RoboDK station: AmbienteRecriado.rdk

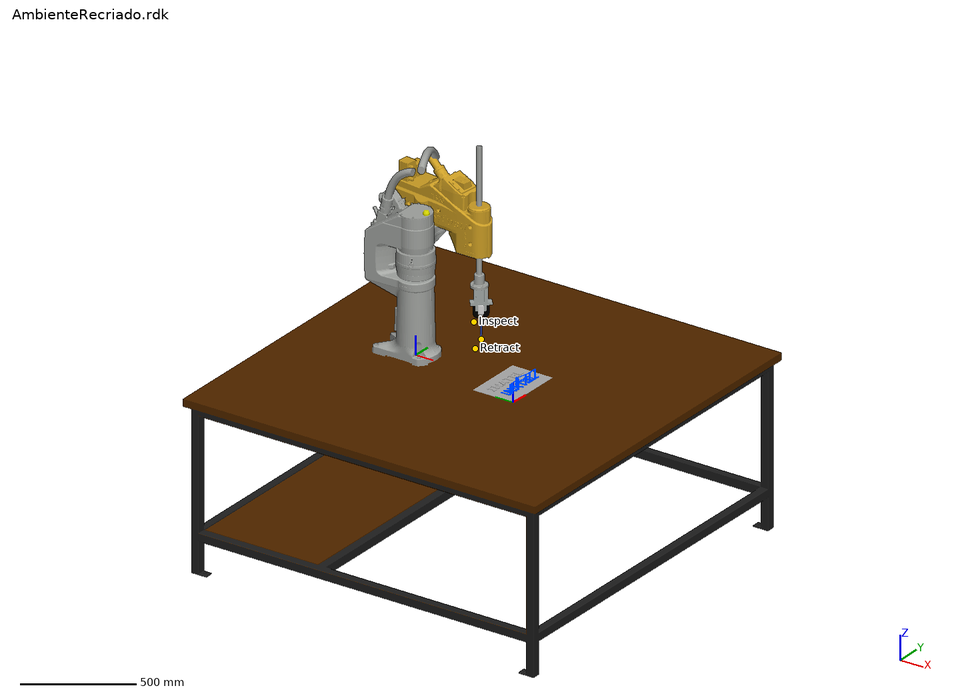
[picture v0: the station drawn from its stored meshes, robots at their saved joint values, targets as dots, program paths as lines]
Station FollowCurves_Inatel (saved by RoboDK 5.5.2). Poses are relative to the parent item; angles as X-Y-Z fixed-axis rotations.
  - frame World at (0, 0, 835) mm
    - robot Staubli TS60 FL 200 (model Staubli TS60 FL 400): 4 axes, payload 2 kg, reach 600 mm, repeatability 0.01 mm, weight 55 kg
        modified DH rows (alpha deg, a mm, theta deg, d mm): 0, 0, 0, 0; 0, 330, 0, 0; 0, 270, 0, 170 linear; 180, 0, 0, 0
        joint limits [-140, -150, 0, -500] to [140, 150, 200, 500]; home [0, 0, 0, 0]; saved at [112.244, -119.359, 90, 172.885]
      - tool GarraCompleta, TCP at (0, 0, 200) mm, size 97 x 40 x 153.1 mm, geometry from GarraCompleta.STL
        - object Suporte_e_Caneta at (4.39, 18.92, -137) mm, rotated rx 0 ry 0 rz 48 deg, size 26 x 26 x 165.9 mm, geometry from Suporte_e_Caneta.STL
      - tool TCP_Garra, TCP at (0, 17, 260) mm
    - frame Reference SW at (610, -140, 0) mm, rotated rx 0 ry 0 rz 90 deg
      - object SWPart at (0, 0, 0) mm, size 295 x 210 x 6 mm, geometry from SWPart.stl
    - target Retract (Cartesian target) at (261.87, 75.71, 73.19) mm, rotated rx -180 ry 0 rz 180 deg; joints [65.057, -128.028, 163.19, 117.03] of Staubli TS60 FL 200
    - target Inspect (Cartesian target) at (104.05, 290.73, 73.19) mm, rotated rx -180 ry 0 rz -180 deg; joints [120.14, -122.614, 163.19, 177.527] of Staubli TS60 FL 200
    - target Peça (Cartesian target) at (143, 289, 0) mm, rotated rx -180 ry 0 rz -180 deg; joints [120.14, -122.614, 163.19, 177.527] of Staubli TS60 FL 200
    - target Encaixe (Cartesian target) at (143, 289, 0) mm, rotated rx -180 ry 0 rz -180 deg; joints [120.14, -122.614, 163.19, 177.527] of Staubli TS60 FL 200
  - object Mesa at (350, 0, 0) mm, size 1850 x 1850 x 835 mm, geometry from Mesa.STL
  - program Attach (1 instructions, listed below)
  - machining project Path1 settings: rotZ(0) | rotX(0)*rotY(0) | rotz(0) | onStart | onPathStart | onApproach | onPoint | onRetract | onFinish | SetRPM(%1) | SetTool(%1) | Extruder(%1) | default | default | OutOnMov(%1) | OutOffMov(%1) | onPathFinish | M_RunCode(%1)
  - program Path1 (314 instructions, listed below)
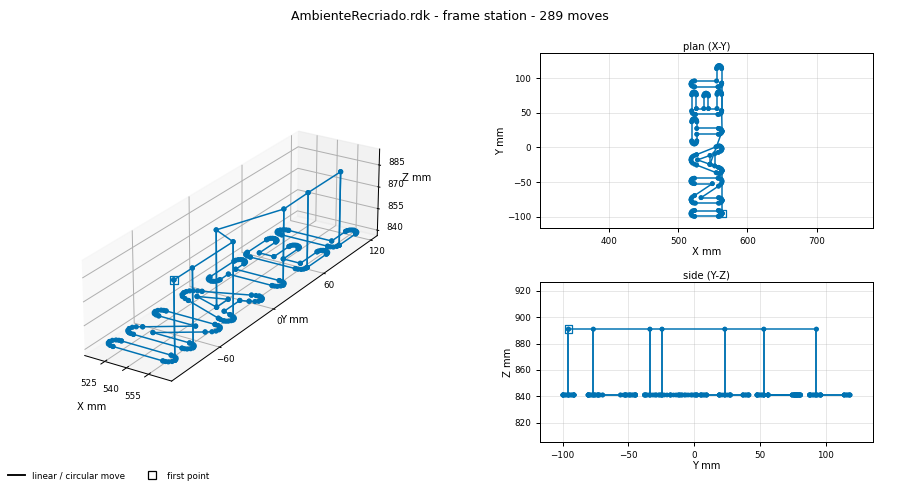
[picture p0: tool path of AmbienteRecriado.rdk in frame station, 289 of 289 moves have a stored position in this frame; points joined in program order, loops and branches not executed]

--- program Attach (robot Staubli TS60 FL 200) ---
  Attach to GarraCompleta

--- program Path1 (robot Staubli TS60 FL 200) ---
  Smooth(1)
  Set speed (1000.0 mm/s)
  Set Ref.: Reference SW
  Set Tool: TCP_Garra
  Show TCP_Garra
  MoveJ 1 to (44.52, 46.68, 56) mm, rotated rx -180 ry 0 rz 90 deg; joints [3.841, -33.741, 146, 150.101]
  MoveL 2 to (44.52, 46.68, 56) mm, rotated rx -180 ry 0 rz 90 deg; joints [3.841, -33.741, 146, 150.101]
  MoveL 3 to (44.52, 46.68, 6) mm, rotated rx -180 ry 0 rz 90 deg; joints [3.841, -33.741, 96, 150.101]
  MoveL 4 to (44.52, 46.68, 6) mm, rotated rx -180 ry 0 rz 90 deg; joints [3.841, -33.741, 96, 150.101]
  Set speed (50.0 mm/s)
  MoveL 5 to (42.47, 47.22, 6) mm, rotated rx -180 ry 0 rz 90 deg; joints [3.667, -33.825, 96, 149.843]
  MoveL 6 to (41.01, 48.77, 6) mm, rotated rx -180 ry 0 rz 90 deg; joints [3.851, -34.627, 96, 149.224]
  MoveL 7 to (40.48, 50.37, 6) mm, rotated rx -180 ry 0 rz 90 deg; joints [4.183, -35.562, 96, 148.621]
  MoveL 8 to (40.34, 52.05, 6) mm, rotated rx -180 ry 0 rz 90 deg; joints [4.583, -36.569, 96, 148.014]
  MoveL 9 to (40.34, 52.05, 6) mm, rotated rx -180 ry 0 rz 90 deg; joints [4.583, -36.569, 96, 148.014]
  MoveL 10 to (40.34, 86.33, 6) mm, rotated rx -180 ry 0 rz 90 deg; joints [11.299, -53.485, 96, 137.814]
  MoveL 11 to (40.34, 86.33, 6) mm, rotated rx -180 ry 0 rz 90 deg; joints [11.299, -53.485, 96, 137.814]
  MoveL 12 to (40.58, 88.46, 6) mm, rotated rx -180 ry 0 rz 90 deg; joints [11.67, -54.391, 96, 137.279]
  MoveL 13 to (41.53, 90.37, 6) mm, rotated rx -180 ry 0 rz 90 deg; joints [12.104, -55.258, 96, 136.846]
  MoveL 14 to (42.87, 91.36, 6) mm, rotated rx -180 ry 0 rz 90 deg; joints [12.451, -55.78, 96, 136.67]
  MoveL 15 to (44.52, 91.68, 6) mm, rotated rx -180 ry 0 rz 90 deg; joints [12.736, -56.054, 96, 136.682]
  MoveL 16 to (44.52, 91.68, 6) mm, rotated rx -180 ry 0 rz 90 deg; joints [12.736, -56.054, 96, 136.682]
  MoveL 17 to (46.6, 91.17, 6) mm, rotated rx -180 ry 0 rz 90 deg; joints [12.956, -56.028, 96, 136.929]
  MoveL 18 to (48.1, 89.64, 6) mm, rotated rx -180 ry 0 rz 90 deg; joints [12.935, -55.538, 96, 137.397]
  MoveL 19 to (48.65, 88.03, 6) mm, rotated rx -180 ry 0 rz 90 deg; joints [12.762, -54.929, 96, 137.833]
  MoveL 20 to (48.78, 86.33, 6) mm, rotated rx -180 ry 0 rz 90 deg; joints [12.512, -54.24, 96, 138.272]
  MoveL 21 to (48.78, 86.33, 6) mm, rotated rx -180 ry 0 rz 90 deg; joints [12.512, -54.24, 96, 138.272]
  MoveL 22 to (48.78, 52.05, 6) mm, rotated rx -180 ry 0 rz 90 deg; joints [5.865, -37.581, 96, 148.284]
  MoveL 23 to (48.78, 52.05, 6) mm, rotated rx -180 ry 0 rz 90 deg; joints [5.865, -37.581, 96, 148.284]
  MoveL 24 to (48.55, 49.89, 6) mm, rotated rx -180 ry 0 rz 90 deg; joints [5.298, -36.265, 96, 149.033]
  MoveL 25 to (47.57, 47.97, 6) mm, rotated rx -180 ry 0 rz 90 deg; joints [4.657, -34.958, 96, 149.699]
  MoveL 26 to (46.19, 46.99, 6) mm, rotated rx -180 ry 0 rz 90 deg; joints [4.184, -34.157, 96, 150.027]
  MoveL 27 to (44.52, 46.68, 6) mm, rotated rx -180 ry 0 rz 90 deg; joints [3.841, -33.741, 96, 150.101]
  Set speed (1000.0 mm/s)
  MoveL 28 to (44.52, 46.68, 6) mm, rotated rx -180 ry 0 rz 90 deg; joints [3.841, -33.741, 96, 150.101]
  MoveL 29 to (44.52, 46.68, 56) mm, rotated rx -180 ry 0 rz 90 deg; joints [3.841, -33.741, 146, 150.101]
  Set speed (1000.0 mm/s)
  MoveL 30 to (63.41, 46.68, 56) mm, rotated rx -180 ry 0 rz 90 deg; joints [6.675, -35.932, 146, 150.744]
  MoveL 31 to (63.41, 46.68, 6) mm, rotated rx -180 ry 0 rz 90 deg; joints [6.675, -35.932, 96, 150.744]
  MoveL 32 to (63.41, 46.68, 6) mm, rotated rx -180 ry 0 rz 90 deg; joints [6.675, -35.932, 96, 150.744]
  Set speed (50.0 mm/s)
  MoveL 33 to (61.47, 47.18, 6) mm, rotated rx -180 ry 0 rz 90 deg; joints [6.523, -36.039, 96, 150.484]
  MoveL 34 to (60.1, 48.64, 6) mm, rotated rx -180 ry 0 rz 90 deg; joints [6.695, -36.785, 96, 149.91]
  MoveL 35 to (59.6, 50.14, 6) mm, rotated rx -180 ry 0 rz 90 deg; joints [6.995, -37.63, 96, 149.365]
  MoveL 36 to (59.47, 51.72, 6) mm, rotated rx -180 ry 0 rz 90 deg; joints [7.358, -38.539, 96, 148.819]
  MoveL 37 to (59.47, 51.72, 6) mm, rotated rx -180 ry 0 rz 90 deg; joints [7.358, -38.539, 96, 148.819]
  MoveL 38 to (59.47, 85.3, 6) mm, rotated rx -180 ry 0 rz 90 deg; joints [13.85, -54.68, 96, 139.171]
  MoveL 39 to (59.47, 85.3, 6) mm, rotated rx -180 ry 0 rz 90 deg; joints [13.85, -54.68, 96, 139.171]
  MoveL 40 to (59.58, 87.2, 6) mm, rotated rx -180 ry 0 rz 90 deg; joints [14.17, -55.47, 96, 138.7]
  MoveL 41 to (59.93, 88.65, 6) mm, rotated rx -180 ry 0 rz 90 deg; joints [14.447, -56.087, 96, 138.36]
  MoveL 42 to (59.93, 88.65, 6) mm, rotated rx -180 ry 0 rz 90 deg; joints [14.447, -56.087, 96, 138.36]
  MoveL 43 to (60.79, 90.01, 6) mm, rotated rx -180 ry 0 rz 90 deg; joints [14.778, -56.697, 96, 138.08]
  MoveL 44 to (62.05, 91.02, 6) mm, rotated rx -180 ry 0 rz 90 deg; joints [15.107, -57.19, 96, 137.917]
  MoveL 45 to (64.47, 91.68, 6) mm, rotated rx -180 ry 0 rz 90 deg; joints [15.542, -57.625, 96, 137.918]
  MoveL 46 to (64.47, 91.68, 6) mm, rotated rx -180 ry 0 rz 90 deg; joints [15.542, -57.625, 96, 137.918]
  MoveL 47 to (66.75, 91.13, 6) mm, rotated rx -180 ry 0 rz 90 deg; joints [15.773, -57.568, 96, 138.204]
  MoveL 48 to (68.49, 89.54, 6) mm, rotated rx -180 ry 0 rz 90 deg; joints [15.764, -57.054, 96, 138.71]
  MoveL 49 to (70.49, 86.4, 6) mm, rotated rx -180 ry 0 rz 90 deg; joints [15.541, -55.923, 96, 139.618]
  MoveL 50 to (70.49, 86.4, 6) mm, rotated rx -180 ry 0 rz 90 deg; joints [15.541, -55.923, 96, 139.618]
  MoveL 51 to (87.59, 60.74, 6) mm, rotated rx -180 ry 0 rz 90 deg; joints [13.186, -45.589, 96, 147.597]
  MoveL 52 to (87.59, 60.74, 6) mm, rotated rx -180 ry 0 rz 90 deg; joints [13.186, -45.589, 96, 147.597]
  MoveL 53 to (87.59, 86.63, 6) mm, rotated rx -180 ry 0 rz 90 deg; joints [17.859, -57.048, 96, 140.811]
  MoveL 54 to (87.59, 86.63, 6) mm, rotated rx -180 ry 0 rz 90 deg; joints [17.859, -57.048, 96, 140.811]
  MoveL 55 to (87.81, 88.64, 6) mm, rotated rx -180 ry 0 rz 90 deg; joints [18.205, -57.858, 96, 140.348]
  MoveL 56 to (88.67, 90.44, 6) mm, rotated rx -180 ry 0 rz 90 deg; joints [18.602, -58.614, 96, 139.989]
  MoveL 57 to (89.94, 91.38, 6) mm, rotated rx -180 ry 0 rz 90 deg; joints [18.913, -59.045, 96, 139.869]
  MoveL 58 to (91.49, 91.68, 6) mm, rotated rx -180 ry 0 rz 90 deg; joints [19.161, -59.236, 96, 139.925]
  MoveL 59 to (91.49, 91.68, 6) mm, rotated rx -180 ry 0 rz 90 deg; joints [19.161, -59.236, 96, 139.925]
  MoveL 60 to (93.45, 91.21, 6) mm, rotated rx -180 ry 0 rz 90 deg; joints [19.342, -59.147, 96, 140.195]
  MoveL 61 to (94.84, 89.75, 6) mm, rotated rx -180 ry 0 rz 90 deg; joints [19.294, -58.644, 96, 140.65]
  MoveL 62 to (95.34, 88.23, 6) mm, rotated rx -180 ry 0 rz 90 deg; joints [19.118, -58.07, 96, 141.048]
  MoveL 63 to (95.47, 86.63, 6) mm, rotated rx -180 ry 0 rz 90 deg; joints [18.879, -57.442, 96, 141.437]
  MoveL 64 to (95.47, 86.63, 6) mm, rotated rx -180 ry 0 rz 90 deg; joints [18.879, -57.442, 96, 141.437]
  MoveL 65 to (95.47, 52.41, 6) mm, rotated rx -180 ry 0 rz 90 deg; joints [12.405, -41.776, 96, 150.63]
  MoveL 66 to (95.47, 52.41, 6) mm, rotated rx -180 ry 0 rz 90 deg; joints [12.405, -41.776, 96, 150.63]
  MoveL 67 to (95.22, 50.06, 6) mm, rotated rx -180 ry 0 rz 90 deg; joints [11.832, -40.479, 96, 151.353]
  MoveL 68 to (94.17, 47.96, 6) mm, rotated rx -180 ry 0 rz 90 deg; joints [11.197, -39.232, 96, 151.965]
  MoveL 69 to (92.63, 46.96, 6) mm, rotated rx -180 ry 0 rz 90 deg; joints [10.751, -38.552, 96, 152.199]
  MoveL 70 to (90.8, 46.68, 6) mm, rotated rx -180 ry 0 rz 90 deg; joints [10.443, -38.265, 96, 152.178]
  MoveL 71 to (90.8, 46.68, 6) mm, rotated rx -180 ry 0 rz 90 deg; joints [10.443, -38.265, 96, 152.178]
  MoveL 72 to (88.35, 47.15, 6) mm, rotated rx -180 ry 0 rz 90 deg; joints [10.238, -38.37, 96, 151.868]
  MoveL 73 to (86.36, 48.66, 6) mm, rotated rx -180 ry 0 rz 90 deg; joints [10.344, -39.102, 96, 151.243]
  MoveL 74 to (84.03, 51.85, 6) mm, rotated rx -180 ry 0 rz 90 deg; joints [10.785, -40.719, 96, 150.067]
  MoveL 75 to (84.03, 51.85, 6) mm, rotated rx -180 ry 0 rz 90 deg; joints [10.785, -40.719, 96, 150.067]
  MoveL 76 to (67.34, 77.05, 6) mm, rotated rx -180 ry 0 rz 90 deg; joints [13.558, -51.771, 96, 141.787]
  MoveL 77 to (67.34, 77.05, 6) mm, rotated rx -180 ry 0 rz 90 deg; joints [13.558, -51.771, 96, 141.787]
  MoveL 78 to (67.34, 51.7, 6) mm, rotated rx -180 ry 0 rz 90 deg; joints [8.472, -39.278, 96, 149.194]
  MoveL 79 to (67.34, 51.7, 6) mm, rotated rx -180 ry 0 rz 90 deg; joints [8.472, -39.278, 96, 149.194]
  MoveL 80 to (67.12, 49.7, 6) mm, rotated rx -180 ry 0 rz 90 deg; joints [7.963, -38.108, 96, 149.855]
  MoveL 81 to (66.21, 47.92, 6) mm, rotated rx -180 ry 0 rz 90 deg; joints [7.394, -36.967, 96, 150.427]
  MoveL 82 to (64.95, 46.98, 6) mm, rotated rx -180 ry 0 rz 90 deg; joints [6.976, -36.275, 96, 150.701]
  MoveL 83 to (63.41, 46.68, 6) mm, rotated rx -180 ry 0 rz 90 deg; joints [6.675, -35.932, 96, 150.744]
  Set speed (1000.0 mm/s)
  MoveL 84 to (63.41, 46.68, 6) mm, rotated rx -180 ry 0 rz 90 deg; joints [6.675, -35.932, 96, 150.744]
  MoveL 85 to (63.41, 46.68, 56) mm, rotated rx -180 ry 0 rz 90 deg; joints [6.675, -35.932, 146, 150.744]
  Set speed (1000.0 mm/s)
  MoveL 86 to (106.38, 46.68, 56) mm, rotated rx -180 ry 0 rz 90 deg; joints [12.427, -39.201, 146, 153.226]
  MoveL 87 to (106.38, 46.68, 6) mm, rotated rx -180 ry 0 rz 90 deg; joints [12.427, -39.201, 96, 153.226]
  MoveL 88 to (106.38, 46.68, 6) mm, rotated rx -180 ry 0 rz 90 deg; joints [12.427, -39.201, 96, 153.226]
  Set speed (50.0 mm/s)
  MoveL 89 to (104.66, 47.06, 6) mm, rotated rx -180 ry 0 rz 90 deg; joints [12.307, -39.332, 96, 152.975]
  MoveL 90 to (103.24, 48.13, 6) mm, rotated rx -180 ry 0 rz 90 deg; joints [12.388, -39.858, 96, 152.529]
  MoveL 91 to (102.49, 49.3, 6) mm, rotated rx -180 ry 0 rz 90 deg; joints [12.572, -40.472, 96, 152.1]
  MoveL 92 to (102.22, 50.66, 6) mm, rotated rx -180 ry 0 rz 90 deg; joints [12.858, -41.208, 96, 151.649]
  MoveL 93 to (102.22, 50.66, 6) mm, rotated rx -180 ry 0 rz 90 deg; joints [12.858, -41.208, 96, 151.649]
  MoveL 94 to (102.76, 53.21, 6) mm, rotated rx -180 ry 0 rz 90 deg; joints [13.507, -42.609, 96, 150.898]
  MoveL 95 to (103.48, 55.14, 6) mm, rotated rx -180 ry 0 rz 90 deg; joints [14.024, -43.654, 96, 150.37]
  MoveL 96 to (103.48, 55.14, 6) mm, rotated rx -180 ry 0 rz 90 deg; joints [14.024, -43.654, 96, 150.37]
  MoveL 97 to (114.5, 83.4, 6) mm, rotated rx -180 ry 0 rz 90 deg; joints [20.734, -56.9, 96, 143.834]
  MoveL 98 to (114.5, 83.4, 6) mm, rotated rx -180 ry 0 rz 90 deg; joints [20.734, -56.9, 96, 143.834]
  MoveL 99 to (115.72, 86.57, 6) mm, rotated rx -180 ry 0 rz 90 deg; joints [21.408, -58.207, 96, 143.201]
  MoveL 100 to (117.32, 89.55, 6) mm, rotated rx -180 ry 0 rz 90 deg; joints [22.087, -59.427, 96, 142.66]
  MoveL 101 to (119.41, 91.18, 6) mm, rotated rx -180 ry 0 rz 90 deg; joints [22.602, -60.117, 96, 142.485]
  MoveL 102 to (122.01, 91.68, 6) mm, rotated rx -180 ry 0 rz 90 deg; joints [22.997, -60.377, 96, 142.62]
  MoveL 103 to (122.01, 91.68, 6) mm, rotated rx -180 ry 0 rz 90 deg; joints [22.997, -60.377, 96, 142.62]
  MoveL 104 to (124.24, 91.34, 6) mm, rotated rx -180 ry 0 rz 90 deg; joints [23.214, -60.304, 96, 142.909]
  MoveL 105 to (126.17, 90.17, 6) mm, rotated rx -180 ry 0 rz 90 deg; joints [23.257, -59.899, 96, 143.359]
  MoveL 106 to (127.53, 88.37, 6) mm, rotated rx -180 ry 0 rz 90 deg; joints [23.127, -59.23, 96, 143.898]
  MoveL 107 to (128.63, 85.94, 6) mm, rotated rx -180 ry 0 rz 90 deg; joints [22.858, -58.299, 96, 144.56]
  MoveL 108 to (129.59, 83.45, 6) mm, rotated rx -180 ry 0 rz 90 deg; joints [22.554, -57.325, 96, 145.228]
  MoveL 109 to (129.59, 83.45, 6) mm, rotated rx -180 ry 0 rz 90 deg; joints [22.554, -57.325, 96, 145.228]
  MoveL 110 to (140.84, 55.38, 6) mm, rotated rx -180 ry 0 rz 90 deg; joints [18.447, -44.973, 96, 153.474]
  MoveL 111 to (140.84, 55.38, 6) mm, rotated rx -180 ry 0 rz 90 deg; joints [18.447, -44.973, 96, 153.474]
  MoveL 112 to (141.77, 52.81, 6) mm, rotated rx -180 ry 0 rz 90 deg; joints [17.977, -43.674, 96, 154.302]
  MoveL 113 to (142.16, 50.71, 6) mm, rotated rx -180 ry 0 rz 90 deg; joints [17.536, -42.576, 96, 154.96]
  MoveL 114 to (142.16, 50.71, 6) mm, rotated rx -180 ry 0 rz 90 deg; joints [17.536, -42.576, 96, 154.96]
  MoveL 115 to (141.7, 48.98, 6) mm, rotated rx -180 ry 0 rz 90 deg; joints [17.079, -41.637, 96, 155.442]
  MoveL 116 to (140.54, 47.6, 6) mm, rotated rx -180 ry 0 rz 90 deg; joints [16.622, -40.864, 96, 155.758]
  MoveL 117 to (139.3, 46.9, 6) mm, rotated rx -180 ry 0 rz 90 deg; joints [16.318, -40.457, 96, 155.861]
  MoveL 118 to (137.9, 46.68, 6) mm, rotated rx -180 ry 0 rz 90 deg; joints [16.109, -40.305, 96, 155.804]
  MoveL 119 to (137.9, 46.68, 6) mm, rotated rx -180 ry 0 rz 90 deg; joints [16.109, -40.305, 96, 155.804]
  MoveL 120 to (135.76, 47.24, 6) mm, rotated rx -180 ry 0 rz 90 deg; joints [16.01, -40.576, 96, 155.434]
  MoveL 121 to (134.31, 48.92, 6) mm, rotated rx -180 ry 0 rz 90 deg; joints [16.251, -41.469, 96, 154.782]
  MoveL 122 to (132.85, 52.12, 6) mm, rotated rx -180 ry 0 rz 90 deg; joints [16.83, -43.147, 96, 153.683]
  MoveL 123 to (132.85, 52.12, 6) mm, rotated rx -180 ry 0 rz 90 deg; joints [16.83, -43.147, 96, 153.683]
  MoveL 124 to (130.79, 57.37, 6) mm, rotated rx -180 ry 0 rz 90 deg; joints [17.755, -45.774, 96, 151.98]
  MoveL 125 to (130.79, 57.37, 6) mm, rotated rx -180 ry 0 rz 90 deg; joints [17.755, -45.774, 96, 151.98]
  MoveL 126 to (113.29, 57.37, 6) mm, rotated rx -180 ry 0 rz 90 deg; joints [15.704, -45.223, 96, 150.482]
  MoveL 127 to (113.29, 57.37, 6) mm, rotated rx -180 ry 0 rz 90 deg; joints [15.704, -45.223, 96, 150.482]
  MoveL 128 to (111.24, 52, 6) mm, rotated rx -180 ry 0 rz 90 deg; joints [14.277, -42.371, 96, 151.906]
  MoveL 129 to (111.24, 52, 6) mm, rotated rx -180 ry 0 rz 90 deg; joints [14.277, -42.371, 96, 151.906]
  MoveL 130 to (110.4, 49.98, 6) mm, rotated rx -180 ry 0 rz 90 deg; joints [13.709, -41.242, 96, 152.467]
  MoveL 131 to (109.38, 48.05, 6) mm, rotated rx -180 ry 0 rz 90 deg; joints [13.126, -40.124, 96, 153.002]
  MoveL 132 to (108.08, 46.96, 6) mm, rotated rx -180 ry 0 rz 90 deg; joints [12.704, -39.446, 96, 153.257]
  MoveL 133 to (106.38, 46.68, 6) mm, rotated rx -180 ry 0 rz 90 deg; joints [12.427, -39.201, 96, 153.226]
  Set speed (1000.0 mm/s)
  MoveL 134 to (106.38, 46.68, 6) mm, rotated rx -180 ry 0 rz 90 deg; joints [12.427, -39.201, 96, 153.226]
  MoveL 135 to (106.38, 46.68, 56) mm, rotated rx -180 ry 0 rz 90 deg; joints [12.427, -39.201, 146, 153.226]
  Set speed (1000.0 mm/s)
  MoveL 136 to (115.58, 64.12, 56) mm, rotated rx -180 ry 0 rz 90 deg; joints [17.364, -48.574, 146, 148.79]
  MoveL 137 to (115.58, 64.12, 6) mm, rotated rx -180 ry 0 rz 90 deg; joints [17.364, -48.574, 96, 148.79]
  MoveL 138 to (115.58, 64.12, 6) mm, rotated rx -180 ry 0 rz 90 deg; joints [17.364, -48.574, 96, 148.79]
  Set speed (50.0 mm/s)
  MoveL 139 to (121.95, 82.12, 6) mm, rotated rx -180 ry 0 rz 90 deg; joints [21.42, -56.602, 96, 144.818]
  MoveL 140 to (121.95, 82.12, 6) mm, rotated rx -180 ry 0 rz 90 deg; joints [21.42, -56.602, 96, 144.818]
  MoveL 141 to (128.45, 64.12, 6) mm, rotated rx -180 ry 0 rz 90 deg; joints [18.878, -48.959, 96, 149.919]
  MoveL 142 to (128.45, 64.12, 6) mm, rotated rx -180 ry 0 rz 90 deg; joints [18.878, -48.959, 96, 149.919]
  MoveL 143 to (115.58, 64.12, 6) mm, rotated rx -180 ry 0 rz 90 deg; joints [17.364, -48.574, 96, 148.79]
  Set speed (1000.0 mm/s)
  MoveL 144 to (115.58, 64.12, 6) mm, rotated rx -180 ry 0 rz 90 deg; joints [17.364, -48.574, 96, 148.79]
  MoveL 145 to (115.58, 64.12, 56) mm, rotated rx -180 ry 0 rz 90 deg; joints [17.364, -48.574, 146, 148.79]
  Set speed (1000.0 mm/s)
  MoveL 146 to (163.28, 46.68, 56) mm, rotated rx -180 ry 0 rz 90 deg; joints [18.761, -40.467, 146, 158.294]
  MoveL 147 to (163.28, 46.68, 6) mm, rotated rx -180 ry 0 rz 90 deg; joints [18.761, -40.467, 96, 158.294]
  MoveL 148 to (163.28, 46.68, 6) mm, rotated rx -180 ry 0 rz 90 deg; joints [18.761, -40.467, 96, 158.294]
  Set speed (50.0 mm/s)
  MoveL 149 to (161.21, 47.19, 6) mm, rotated rx -180 ry 0 rz 90 deg; joints [18.681, -40.762, 96, 157.92]
  MoveL 150 to (159.71, 48.7, 6) mm, rotated rx -180 ry 0 rz 90 deg; joints [18.901, -41.598, 96, 157.302]
  MoveL 151 to (159.17, 50.3, 6) mm, rotated rx -180 ry 0 rz 90 deg; joints [19.228, -42.461, 96, 156.767]
  MoveL 152 to (159.03, 51.99, 6) mm, rotated rx -180 ry 0 rz 90 deg; joints [19.607, -43.35, 96, 156.258]
  MoveL 153 to (159.03, 51.99, 6) mm, rotated rx -180 ry 0 rz 90 deg; joints [19.607, -43.35, 96, 156.258]
  MoveL 154 to (159.03, 83.24, 6) mm, rotated rx -180 ry 0 rz 90 deg; joints [25.842, -57.526, 96, 148.316]
  MoveL 155 to (159.03, 83.24, 6) mm, rotated rx -180 ry 0 rz 90 deg; joints [25.842, -57.526, 96, 148.316]
  MoveL 156 to (149.42, 83.24, 6) mm, rotated rx -180 ry 0 rz 90 deg; joints [24.787, -57.505, 96, 147.282]
  MoveL 157 to (149.42, 83.24, 6) mm, rotated rx -180 ry 0 rz 90 deg; joints [24.787, -57.505, 96, 147.282]
  MoveL 158 to (147.61, 83.45, 6) mm, rotated rx -180 ry 0 rz 90 deg; joints [24.622, -57.578, 96, 147.044]
  MoveL 159 to (146.01, 84.29, 6) mm, rotated rx -180 ry 0 rz 90 deg; joints [24.588, -57.903, 96, 146.685]
  MoveL 160 to (145.21, 85.47, 6) mm, rotated rx -180 ry 0 rz 90 deg; joints [24.699, -58.365, 96, 146.334]
  MoveL 161 to (144.97, 86.88, 6) mm, rotated rx -180 ry 0 rz 90 deg; joints [24.908, -58.917, 96, 145.991]
  MoveL 162 to (144.97, 86.88, 6) mm, rotated rx -180 ry 0 rz 90 deg; joints [24.908, -58.917, 96, 145.991]
  MoveL 163 to (145.37, 88.65, 6) mm, rotated rx -180 ry 0 rz 90 deg; joints [25.25, -59.612, 96, 145.638]
  MoveL 164 to (146.64, 89.94, 6) mm, rotated rx -180 ry 0 rz 90 deg; joints [25.607, -60.122, 96, 145.485]
  MoveL 165 to (147.99, 90.43, 6) mm, rotated rx -180 ry 0 rz 90 deg; joints [25.84, -60.319, 96, 145.521]
  MoveL 166 to (149.42, 90.55, 6) mm, rotated rx -180 ry 0 rz 90 deg; joints [26.023, -60.377, 96, 145.646]
  MoveL 167 to (149.42, 90.55, 6) mm, rotated rx -180 ry 0 rz 90 deg; joints [26.023, -60.377, 96, 145.646]
  MoveL 168 to (177.08, 90.55, 6) mm, rotated rx -180 ry 0 rz 90 deg; joints [29.017, -60.249, 96, 148.768]
  MoveL 169 to (177.08, 90.55, 6) mm, rotated rx -180 ry 0 rz 90 deg; joints [29.017, -60.249, 96, 148.768]
  MoveL 170 to (178.9, 90.35, 6) mm, rotated rx -180 ry 0 rz 90 deg; joints [29.17, -60.141, 96, 149.03]
  MoveL 171 to (180.52, 89.49, 6) mm, rotated rx -180 ry 0 rz 90 deg; joints [29.188, -59.782, 96, 149.406]
  MoveL 172 to (181.33, 88.3, 6) mm, rotated rx -180 ry 0 rz 90 deg; joints [29.064, -59.306, 96, 149.759]
  MoveL 173 to (181.58, 86.88, 6) mm, rotated rx -180 ry 0 rz 90 deg; joints [28.841, -58.745, 96, 150.097]
  MoveL 174 to (181.58, 86.88, 6) mm, rotated rx -180 ry 0 rz 90 deg; joints [28.841, -58.745, 96, 150.097]
  MoveL 175 to (181.16, 85.11, 6) mm, rotated rx -180 ry 0 rz 90 deg; joints [28.485, -58.053, 96, 150.433]
  MoveL 176 to (179.87, 83.83, 6) mm, rotated rx -180 ry 0 rz 90 deg; joints [28.127, -57.564, 96, 150.563]
  MoveL 177 to (178.51, 83.36, 6) mm, rotated rx -180 ry 0 rz 90 deg; joints [27.905, -57.4, 96, 150.505]
  MoveL 178 to (177.08, 83.24, 6) mm, rotated rx -180 ry 0 rz 90 deg; joints [27.737, -57.373, 96, 150.364]
  MoveL 179 to (177.08, 83.24, 6) mm, rotated rx -180 ry 0 rz 90 deg; joints [27.737, -57.373, 96, 150.364]
  MoveL 180 to (167.47, 83.24, 6) mm, rotated rx -180 ry 0 rz 90 deg; joints [26.742, -57.485, 96, 149.257]
  MoveL 181 to (167.47, 83.24, 6) mm, rotated rx -180 ry 0 rz 90 deg; joints [26.742, -57.485, 96, 149.257]
  MoveL 182 to (167.47, 51.99, 6) mm, rotated rx -180 ry 0 rz 90 deg; joints [20.452, -43.3, 96, 157.152]
  MoveL 183 to (167.47, 51.99, 6) mm, rotated rx -180 ry 0 rz 90 deg; joints [20.452, -43.3, 96, 157.152]
  MoveL 184 to (167.24, 49.86, 6) mm, rotated rx -180 ry 0 rz 90 deg; joints [19.927, -42.176, 96, 157.751]
  MoveL 185 to (166.28, 47.96, 6) mm, rotated rx -180 ry 0 rz 90 deg; joints [19.373, -41.154, 96, 158.219]
  MoveL 186 to (164.92, 46.99, 6) mm, rotated rx -180 ry 0 rz 90 deg; joints [19, -40.627, 96, 158.373]
  MoveL 187 to (163.28, 46.68, 6) mm, rotated rx -180 ry 0 rz 90 deg; joints [18.761, -40.467, 96, 158.294]
  Set speed (1000.0 mm/s)
  MoveL 188 to (163.28, 46.68, 6) mm, rotated rx -180 ry 0 rz 90 deg; joints [18.761, -40.467, 96, 158.294]
  MoveL 189 to (163.28, 46.68, 56) mm, rotated rx -180 ry 0 rz 90 deg; joints [18.761, -40.467, 146, 158.294]
  Set speed (1000.0 mm/s)
  MoveL 190 to (192.89, 47.24, 56) mm, rotated rx -180 ry 0 rz 90 deg; joints [21.636, -40.161, 146, 161.475]
  MoveL 191 to (192.89, 47.24, 6) mm, rotated rx -180 ry 0 rz 90 deg; joints [21.636, -40.161, 96, 161.475]
  MoveL 192 to (192.89, 47.24, 6) mm, rotated rx -180 ry 0 rz 90 deg; joints [21.636, -40.161, 96, 161.475]
  Set speed (50.0 mm/s)
  MoveL 193 to (191.28, 47.37, 6) mm, rotated rx -180 ry 0 rz 90 deg; joints [21.53, -40.29, 96, 161.241]
  MoveL 194 to (189.75, 47.88, 6) mm, rotated rx -180 ry 0 rz 90 deg; joints [21.527, -40.626, 96, 160.902]
  MoveL 195 to (188.57, 48.96, 6) mm, rotated rx -180 ry 0 rz 90 deg; joints [21.693, -41.256, 96, 160.436]
  MoveL 196 to (187.89, 50.73, 6) mm, rotated rx -180 ry 0 rz 90 deg; joints [22.066, -42.233, 96, 159.833]
  MoveL 197 to (187.72, 52.62, 6) mm, rotated rx -180 ry 0 rz 90 deg; joints [22.505, -43.24, 96, 159.265]
  MoveL 198 to (187.72, 52.62, 6) mm, rotated rx -180 ry 0 rz 90 deg; joints [22.505, -43.24, 96, 159.265]
  MoveL 199 to (187.72, 85.17, 6) mm, rotated rx -180 ry 0 rz 90 deg; joints [29.152, -57.941, 96, 151.21]
  MoveL 200 to (187.72, 85.17, 6) mm, rotated rx -180 ry 0 rz 90 deg; joints [29.152, -57.941, 96, 151.21]
  MoveL 201 to (188, 87.57, 6) mm, rotated rx -180 ry 0 rz 90 deg; joints [29.607, -58.883, 96, 150.725]
  MoveL 202 to (189.28, 89.59, 6) mm, rotated rx -180 ry 0 rz 90 deg; joints [30.088, -59.639, 96, 150.449]
  MoveL 203 to (191, 90.36, 6) mm, rotated rx -180 ry 0 rz 90 deg; joints [30.394, -59.897, 96, 150.497]
  MoveL 204 to (192.89, 90.55, 6) mm, rotated rx -180 ry 0 rz 90 deg; joints [30.613, -59.921, 96, 150.693]
  MoveL 205 to (192.89, 90.55, 6) mm, rotated rx -180 ry 0 rz 90 deg; joints [30.613, -59.921, 96, 150.693]
  MoveL 206 to (216, 90.55, 6) mm, rotated rx -180 ry 0 rz 90 deg; joints [32.787, -59.102, 96, 153.684]
  MoveL 207 to (216, 90.55, 6) mm, rotated rx -180 ry 0 rz 90 deg; joints [32.787, -59.102, 96, 153.684]
  MoveL 208 to (217.68, 90.37, 6) mm, rotated rx -180 ry 0 rz 90 deg; joints [32.903, -58.955, 96, 153.948]
  MoveL 209 to (219.17, 89.59, 6) mm, rotated rx -180 ry 0 rz 90 deg; joints [32.892, -58.58, 96, 154.312]
  MoveL 210 to (219.93, 88.5, 6) mm, rotated rx -180 ry 0 rz 90 deg; joints [32.759, -58.117, 96, 154.642]
  MoveL 211 to (220.16, 87.2, 6) mm, rotated rx -180 ry 0 rz 90 deg; joints [32.537, -57.589, 96, 154.948]
  MoveL 212 to (220.16, 87.2, 6) mm, rotated rx -180 ry 0 rz 90 deg; joints [32.537, -57.589, 96, 154.948]
  MoveL 213 to (219.78, 85.55, 6) mm, rotated rx -180 ry 0 rz 90 deg; joints [32.196, -56.948, 96, 155.248]
  MoveL 214 to (218.6, 84.35, 6) mm, rotated rx -180 ry 0 rz 90 deg; joints [31.867, -56.519, 96, 155.347]
  MoveL 215 to (217.34, 83.91, 6) mm, rotated rx -180 ry 0 rz 90 deg; joints [31.675, -56.403, 96, 155.272]
  MoveL 216 to (216, 83.8, 6) mm, rotated rx -180 ry 0 rz 90 deg; joints [31.537, -56.419, 96, 155.118]
  MoveL 217 to (216, 83.8, 6) mm, rotated rx -180 ry 0 rz 90 deg; joints [31.537, -56.419, 96, 155.118]
  MoveL 218 to (196.16, 83.8, 6) mm, rotated rx -180 ry 0 rz 90 deg; joints [29.721, -57.168, 96, 152.553]
  MoveL 219 to (196.16, 83.8, 6) mm, rotated rx -180 ry 0 rz 90 deg; joints [29.721, -57.168, 96, 152.553]
  MoveL 220 to (196.16, 73.12, 6) mm, rotated rx -180 ry 0 rz 90 deg; joints [27.687, -52.704, 96, 154.984]
  MoveL 221 to (196.16, 73.12, 6) mm, rotated rx -180 ry 0 rz 90 deg; joints [27.687, -52.704, 96, 154.984]
  MoveL 222 to (214.43, 73.12, 6) mm, rotated rx -180 ry 0 rz 90 deg; joints [29.307, -51.987, 96, 157.321]
  MoveL 223 to (214.43, 73.12, 6) mm, rotated rx -180 ry 0 rz 90 deg; joints [29.307, -51.987, 96, 157.321]
  MoveL 224 to (216.07, 72.92, 6) mm, rotated rx -180 ry 0 rz 90 deg; joints [29.407, -51.824, 96, 157.583]
  MoveL 225 to (217.51, 72.13, 6) mm, rotated rx -180 ry 0 rz 90 deg; joints [29.365, -51.403, 96, 157.962]
  MoveL 226 to (218.22, 71.05, 6) mm, rotated rx -180 ry 0 rz 90 deg; joints [29.2, -50.887, 96, 158.314]
  MoveL 227 to (218.44, 69.77, 6) mm, rotated rx -180 ry 0 rz 90 deg; joints [28.95, -50.301, 96, 158.649]
  MoveL 228 to (218.44, 69.77, 6) mm, rotated rx -180 ry 0 rz 90 deg; joints [28.95, -50.301, 96, 158.649]
  MoveL 229 to (218.08, 68.15, 6) mm, rotated rx -180 ry 0 rz 90 deg; joints [28.579, -49.585, 96, 158.994]
  MoveL 230 to (216.96, 66.94, 6) mm, rotated rx -180 ry 0 rz 90 deg; joints [28.228, -49.084, 96, 159.144]
  MoveL 231 to (215.73, 66.48, 6) mm, rotated rx -180 ry 0 rz 90 deg; joints [28.03, -48.935, 96, 159.095]
  MoveL 232 to (214.43, 66.37, 6) mm, rotated rx -180 ry 0 rz 90 deg; joints [27.897, -48.946, 96, 158.951]
  MoveL 233 to (214.43, 66.37, 6) mm, rotated rx -180 ry 0 rz 90 deg; joints [27.897, -48.946, 96, 158.951]
  MoveL 234 to (196.16, 66.37, 6) mm, rotated rx -180 ry 0 rz 90 deg; joints [26.316, -49.694, 96, 156.621]
  MoveL 235 to (196.16, 66.37, 6) mm, rotated rx -180 ry 0 rz 90 deg; joints [26.316, -49.694, 96, 156.621]
  MoveL 236 to (196.16, 53.99, 6) mm, rotated rx -180 ry 0 rz 90 deg; joints [23.572, -43.678, 96, 159.894]
  MoveL 237 to (196.16, 53.99, 6) mm, rotated rx -180 ry 0 rz 90 deg; joints [23.572, -43.678, 96, 159.894]
  MoveL 238 to (216.69, 53.99, 6) mm, rotated rx -180 ry 0 rz 90 deg; joints [25.25, -42.725, 96, 162.525]
  MoveL 239 to (216.69, 53.99, 6) mm, rotated rx -180 ry 0 rz 90 deg; joints [25.25, -42.725, 96, 162.525]
  MoveL 240 to (218.38, 53.8, 6) mm, rotated rx -180 ry 0 rz 90 deg; joints [25.332, -42.525, 96, 162.807]
  MoveL 241 to (219.88, 53, 6) mm, rotated rx -180 ry 0 rz 90 deg; joints [25.249, -42.013, 96, 163.235]
  MoveL 242 to (220.64, 51.9, 6) mm, rotated rx -180 ry 0 rz 90 deg; joints [25.03, -41.375, 96, 163.655]
  MoveL 243 to (220.87, 50.59, 6) mm, rotated rx -180 ry 0 rz 90 deg; joints [24.713, -40.64, 96, 164.073]
  MoveL 244 to (220.87, 50.59, 6) mm, rotated rx -180 ry 0 rz 90 deg; joints [24.713, -40.64, 96, 164.073]
  MoveL 245 to (220.47, 48.96, 6) mm, rotated rx -180 ry 0 rz 90 deg; joints [24.262, -39.758, 96, 164.504]
  MoveL 246 to (219.27, 47.79, 6) mm, rotated rx -180 ry 0 rz 90 deg; joints [23.867, -39.168, 96, 164.698]
  MoveL 247 to (218.01, 47.36, 6) mm, rotated rx -180 ry 0 rz 90 deg; joints [23.66, -38.999, 96, 164.661]
  MoveL 248 to (216.69, 47.24, 6) mm, rotated rx -180 ry 0 rz 90 deg; joints [23.532, -39.013, 96, 164.519]
  MoveL 249 to (216.69, 47.24, 6) mm, rotated rx -180 ry 0 rz 90 deg; joints [23.532, -39.013, 96, 164.519]
  MoveL 250 to (192.89, 47.24, 6) mm, rotated rx -180 ry 0 rz 90 deg; joints [21.636, -40.161, 96, 161.475]
  Set speed (1000.0 mm/s)
  MoveL 251 to (192.89, 47.24, 6) mm, rotated rx -180 ry 0 rz 90 deg; joints [21.636, -40.161, 96, 161.475]
  MoveL 252 to (192.89, 47.24, 56) mm, rotated rx -180 ry 0 rz 90 deg; joints [21.636, -40.161, 146, 161.475]
  Set speed (1000.0 mm/s)
  MoveL 253 to (232.82, 47.24, 56) mm, rotated rx -180 ry 0 rz 90 deg; joints [24.649, -37.883, 146, 166.767]
  MoveL 254 to (232.82, 47.24, 6) mm, rotated rx -180 ry 0 rz 90 deg; joints [24.649, -37.883, 96, 166.767]
  MoveL 255 to (232.82, 47.24, 6) mm, rotated rx -180 ry 0 rz 90 deg; joints [24.649, -37.883, 96, 166.767]
  Set speed (50.0 mm/s)
  MoveL 256 to (230.43, 47.58, 6) mm, rotated rx -180 ry 0 rz 90 deg; joints [24.584, -38.267, 96, 166.318]
  MoveL 257 to (228.5, 48.99, 6) mm, rotated rx -180 ry 0 rz 90 deg; joints [24.834, -39.223, 96, 165.611]
  MoveL 258 to (227.82, 50.76, 6) mm, rotated rx -180 ry 0 rz 90 deg; joints [25.254, -40.272, 96, 164.981]
  MoveL 259 to (227.66, 52.66, 6) mm, rotated rx -180 ry 0 rz 90 deg; joints [25.729, -41.329, 96, 164.401]
  MoveL 260 to (227.66, 52.66, 6) mm, rotated rx -180 ry 0 rz 90 deg; joints [25.729, -41.329, 96, 164.401]
  MoveL 261 to (227.66, 86.32, 6) mm, rotated rx -180 ry 0 rz 90 deg; joints [33.012, -56.853, 96, 156.159]
  MoveL 262 to (227.66, 86.32, 6) mm, rotated rx -180 ry 0 rz 90 deg; joints [33.012, -56.853, 96, 156.159]
  MoveL 263 to (227.89, 88.45, 6) mm, rotated rx -180 ry 0 rz 90 deg; joints [33.434, -57.693, 96, 155.741]
  MoveL 264 to (228.83, 90.36, 6) mm, rotated rx -180 ry 0 rz 90 deg; joints [33.87, -58.396, 96, 155.474]
  MoveL 265 to (230.18, 91.36, 6) mm, rotated rx -180 ry 0 rz 90 deg; joints [34.169, -58.713, 96, 155.455]
  MoveL 266 to (231.83, 91.68, 6) mm, rotated rx -180 ry 0 rz 90 deg; joints [34.366, -58.745, 96, 155.621]
  MoveL 267 to (231.83, 91.68, 6) mm, rotated rx -180 ry 0 rz 90 deg; joints [34.366, -58.745, 96, 155.621]
  MoveL 268 to (233.92, 91.16, 6) mm, rotated rx -180 ry 0 rz 90 deg; joints [34.445, -58.425, 96, 156.02]
  MoveL 269 to (235.42, 89.63, 6) mm, rotated rx -180 ry 0 rz 90 deg; joints [34.281, -57.733, 96, 156.548]
  MoveL 270 to (235.96, 88.02, 6) mm, rotated rx -180 ry 0 rz 90 deg; joints [34.019, -57.058, 96, 156.961]
  MoveL 271 to (236.09, 86.32, 6) mm, rotated rx -180 ry 0 rz 90 deg; joints [33.705, -56.367, 96, 157.338]
  MoveL 272 to (236.09, 86.32, 6) mm, rotated rx -180 ry 0 rz 90 deg; joints [33.705, -56.367, 96, 157.338]
  MoveL 273 to (236.09, 54.55, 6) mm, rotated rx -180 ry 0 rz 90 deg; joints [26.789, -41.736, 96, 165.053]
  MoveL 274 to (236.09, 54.55, 6) mm, rotated rx -180 ry 0 rz 90 deg; joints [26.789, -41.736, 96, 165.053]
  MoveL 275 to (253.95, 54.55, 6) mm, rotated rx -180 ry 0 rz 90 deg; joints [27.903, -40.194, 96, 167.709]
  MoveL 276 to (253.95, 54.55, 6) mm, rotated rx -180 ry 0 rz 90 deg; joints [27.903, -40.194, 96, 167.709]
  MoveL 277 to (255.75, 54.32, 6) mm, rotated rx -180 ry 0 rz 90 deg; joints [27.943, -39.889, 96, 168.054]
  MoveL 278 to (257.31, 53.43, 6) mm, rotated rx -180 ry 0 rz 90 deg; joints [27.791, -39.231, 96, 168.56]
  MoveL 279 to (258.12, 52.26, 6) mm, rotated rx -180 ry 0 rz 90 deg; joints [27.519, -38.483, 96, 169.035]
  MoveL 280 to (258.37, 50.87, 6) mm, rotated rx -180 ry 0 rz 90 deg; joints [27.146, -37.644, 96, 169.502]
  MoveL 281 to (258.37, 50.87, 6) mm, rotated rx -180 ry 0 rz 90 deg; joints [27.146, -37.644, 96, 169.502]
  MoveL 282 to (257.96, 49.13, 6) mm, rotated rx -180 ry 0 rz 90 deg; joints [26.632, -36.649, 96, 169.982]
  MoveL 283 to (256.7, 47.85, 6) mm, rotated rx -180 ry 0 rz 90 deg; joints [26.2, -36.008, 96, 170.192]
  MoveL 284 to (255.37, 47.37, 6) mm, rotated rx -180 ry 0 rz 90 deg; joints [25.992, -35.856, 96, 170.136]
  MoveL 285 to (253.95, 47.24, 6) mm, rotated rx -180 ry 0 rz 90 deg; joints [25.882, -35.928, 96, 169.954]
  MoveL 286 to (253.95, 47.24, 6) mm, rotated rx -180 ry 0 rz 90 deg; joints [25.882, -35.928, 96, 169.954]
  MoveL 287 to (232.82, 47.24, 6) mm, rotated rx -180 ry 0 rz 90 deg; joints [24.649, -37.883, 96, 166.767]
  Set speed (1000.0 mm/s)
  MoveL 288 to (232.82, 47.24, 6) mm, rotated rx -180 ry 0 rz 90 deg; joints [24.649, -37.883, 96, 166.767]
  MoveL 289 to (232.82, 47.24, 56) mm, rotated rx -180 ry 0 rz 90 deg; joints [24.649, -37.883, 146, 166.767]
